% RSLogix 500 project COUNTER LOGIC_BAK001.RSS, saved by version 8.30.00.16 %
PROJECT "UNTITLED"    % processor: Bul.1763 MicroLogix 1100 Series B %

PROGRAM FILES
  LAD 2   4 rungs

DATA FILES
  O0 OUTPUT  4 elements
  I1 INPUT  6 elements
  S2 STATUS  66 elements
  B3 BINARY  1 elements
  T4 TIMER  1 elements
  C5 COUNTER  1 elements
  R6 CONTROL  1 elements
  N7 INTEGER  1 elements
  F8 FLOAT  1 elements

LADDER 2
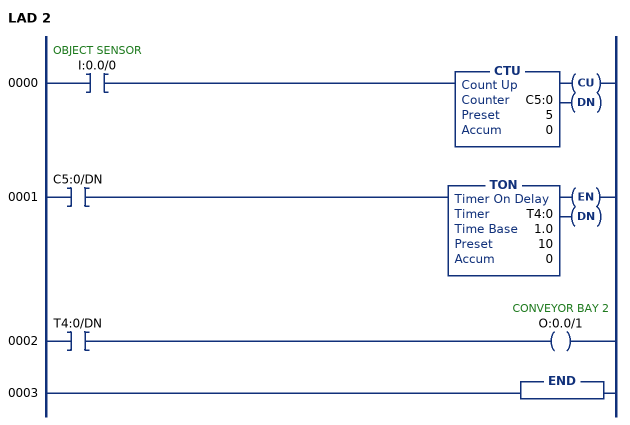
% Rung: 0 %  % edit flag set %
SOR XIC I:0.0/0 CTU C5:0 5 0 EOR
%   I:0.0/0  "OBJECT SENSOR" %
% Rung: 1 %  % edit flag set %
SOR XIC C5:0/DN TON T4:0 1.0 10 0 EOR
% Rung: 2 %  % edit flag set %
SOR XIC T4:0/DN OTE O:0.0/1 EOR
%   O:0.0/1  "CONVEYOR BAY 2" %
% Rung: 3 %
SOR END EOR
